// TIA Portal V17 export
// export: Created 2023-02-13T11:16:35.648872Z, ExportSetting WithDefaults, DisplayName Totally Integrated Automation Portal, DisplayVersion V17, DisplayName TIA Portal Openness, DisplayVersion V17, DisplayName TIA Portal Teamcenter Gateway, DisplayVersion V17, DisplayName TIA Portal Version Control Interface, DisplayVersion V17, DisplayName SINAMICS Startdrive Advanced, DisplayVersion V17, DisplayName SINAMICS Startdrive G130, G150, S120, S150, SINAMICS MV, S210, DisplayVersion V17, DisplayName SINAMICS Startdrive G110M, G120, G120C, G120D, G120P, G115D, DisplayVersion V17, DisplayName STEP 7 Professional, DisplayVersion V17, DisplayName STEP 7 Safety, DisplayVersion V17, DisplayName WinCC Professional, DisplayVersion V17
DATA_BLOCK "IO_Valve_Buffer_DB"   // DB64
VERSION : 0.1
// stored: AutoNumber true, DBAccessibleFromOPCUA true, DBAccessibleFromWebserver true, InstanceOfName IO_Valve_Buffer, InstanceOfType FB
"IO_Valve_Buffer"
   // VAR_INPUT
   //    "lock 1" : Bool;
   //    "lock 2" : Bool;
   //    "lock 3" : Bool;
   //    "lock 4" : Bool;
   //    init : Bool;
   //    reset : Bool;
   //    testing : Bool;
   // END_VAR
   // VAR
   //    "AV-22.11" : "Valve";
   //    "AV-22.21" : "Valve";
   //    "AV-22.22" : "Valve";
   //    "AV-22.23" : "Valve";
   //    "AV-32.01" : "Valve";
   //    "AV-32.02" : "Valve";
   //    "AV-32.03" : "Valve";
   //    "AV-32.04" : "Valve";
   //    "AV-32.11" : "Valve";
   //    "AV-32.21" : "Valve";
   //    "AV-32.22" : "Valve";
   //    "AV-32.23" : "Valve";
   //    "AV-61.01" : "Valve";
   //    "AV-61.02" : "Valve";
   //    "AV-61.03" : "Valve";
   //    "AV-61.04" : "Valve";
   //    "AV-61.05" : "Valve";
   //    "AV-61.21" : "Valve";
   //    "AV-62.06" : "Valve";
   //    "AV-64.01" : "Valve";
   //    "AV-64.02" : "Valve";
   //    "AV-64.03" : "Valve";
   //    "AV-64.04" : "Valve";
   //    "AV-64.05" : "Valve";
   //    "AV-64.06" : "Valve";
   //    "AV-65.01" : "Valve";
   //    "AV-65.02" : "Valve";
   //    "AV-65.03" : "Valve";
   //    "AV-65.04" : "Valve";
   //    "AV-65.05" : "Valve";
   //    "AV-65.21" : "Valve";
   //    "AV-66.01" : "Valve";
   //    "AV-66.02" : "Valve";
   //    "AV-66.03" : "Valve";
   //    "AV-66.04" : "Valve";
   //    "AV-66.05" : "Valve";
   //    "AV-66.06" : "Valve";
   //    "AV-67.01" : "Valve";
   //    "AV-67.02" : "Valve";
   //    "AV-67.03" : "Valve";
   //    "AV-67.04" : "Valve";
   //    "AV-67.05" : "Valve";
   //    "AV-68.01" : "Valve";
   //    "AV-68.02" : "Valve";
   //    "AV-68.03" : "Valve";
   //    "AV-68.04" : "Valve";
   //    "AV-68.05" : "Valve";
   //    "AV-68.06" : "Valve";
   // END_VAR
BEGIN
END_DATA_BLOCK
